{attribute 'GeneratedUsingTerminal: IODEVICETYPE_ETHERCATPROT'}
{attribute addProperty BoxType "IODEVICETYPE_ETHERCATPROT"}
{attribute addProperty Id "Beckhoff_ELXxxxxBeckhoff_ELXxxxx_62AA317A879SyncUnitsSyncUnits_99E584AF18InputsInputs_25A0042B160OutputsOutputs_2397A10E106InfoDataInfoData_E68C61CD28"}
{attribute addProperty CRC "3501359405"}
{attribute addProperty Size "1191"}
TYPE EtherCAT_Master_ELXxxxx_D0B2812D :
STRUCT
	{attribute addProperty Name "Beckhoff ELXxxxx"}
	{attribute addProperty PreviousPort "EtherCAT_Master_ELXxxxx : Master"}
	Beckhoff_ELXxxxx : Beckhoff_ELXxxxx_62AA317A;
	{attribute addProperty Name "SyncUnits"}
	SyncUnits : SyncUnits_99E584AF;
	{attribute addProperty Name "Inputs"}
	Inputs : Inputs_25A0042B;
	{attribute addProperty Name "Outputs"}
	Outputs : Outputs_2397A10E;
	{attribute addProperty Name "InfoData"}
	InfoData : InfoData_E68C61CD;
END_STRUCT
END_TYPE

(* stored: Version 1.2.0.0, ProductVersion 3.1.4024.9
   DUT EtherCAT_Master_ELXxxxx_D0B2812D: Id {4c92e80d-e112-4e48-a73d-bbe4b77d63e3} *)
